FUNCTION TryConvert_WORD_TO_BYTE : BOOL
VAR_INPUT
	in : WORD;
	out : REFERENCE TO BYTE;
END_VAR

IF in > DatatypeLimits.MAX_VALUE_OF_WORD_WHICH_CAN_BE_HELD_IN_A_BYTE THEN
	RETURN;
END_IF

out := WORD_TO_BYTE(in);
TryConvert_WORD_TO_BYTE := TRUE;

END_FUNCTION

(* stored: Version 1.1.0.1, ProductVersion 3.1.4024.12
   POU TryConvert_WORD_TO_BYTE: Id {3fdab202-2d7f-46f2-af29-ad9ca7965189}, SpecialFunc None *)
